// TIA Portal V18 export
DATA_BLOCK "HVAC_Vars"   // DB99
{ S7_Optimized_Access := 'FALSE' }
VERSION : 0.1
// stored: AutoNumber false, DBAccessibleFromOPCUA true, IsOnlyStoredInLoadMemory false, IsWriteProtectedInAS false
   VAR
      Season { S7_SetPoint := 'True'} : "UDT_Store_Season";
      SetPoints { S7_SetPoint := 'True'} : "UDT_Store_Setpoints";
      OpModes { S7_SetPoint := 'True'} : "UDT_Store_OpMode";
      WeekScheduler { S7_SetPoint := 'True'} : "UDT_Store_Scheduler";
      RoomTempSetPointforHMI { S7_SetPoint := 'True'} : Real := 35.0;
      Holidays { S7_SetPoint := 'True'} : Array[1..4] of Date;
      xIsHoliday : Bool := FALSE;
      cDayType : Byte := 16#01;   // 0-WD,1-Mon,2-Cуб,3-Нед,4-Свят
      CurrentDate : Date := D#2026-04-20;
      CurrentTOD : Time_Of_Day := TOD#22:03:20.160;
      iRetVal : Int := 1;
   END_VAR
BEGIN
   Season.cSeasonModeSelection := 16#00;
   Season.cActual := 16#00;   // 0 = Summer 1 = Winter 2 = Midseason, 3=Auro
   Season.cTarget := 16#00;
   Season.cReserve := 16#00;
   Season.rOATtoWinter := 10.0;
   Season.rOATtoSummer := 12.0;
   SetPoints.Room.Actual.rRATHeating := 5.0;
   SetPoints.Room.Actual.rRATCooling := 35.0;
   SetPoints.Room.Actual.rIAQ := 0.0;
   SetPoints.Room.Actual.rBuildingdP := 0.0;
   SetPoints.Room.Comfort.rRATHeating := 18.0;
   SetPoints.Room.Comfort.rRATCooling := 22.0;
   SetPoints.Room.Comfort.rIAQ := 600.0;
   SetPoints.Room.Comfort.rBuildingdP := 5.0;
   SetPoints.Room.PreComfort.rRATHeating := 16.0;
   SetPoints.Room.PreComfort.rRATCooling := 25.0;
   SetPoints.Room.PreComfort.rIAQ := 800.0;
   SetPoints.Room.PreComfort.rBuildingdP := 2.0;
   SetPoints.Room.Econom.rRATHeating := 15.0;
   SetPoints.Room.Econom.rRATCooling := 30.0;
   SetPoints.Room.Econom.rIAQ := 0.0;
   SetPoints.Room.Econom.rBuildingdP := 0.0;
   SetPoints.Room.Protection.rRATHeating := 5.0;
   SetPoints.Room.Protection.rRATCooling := 35.0;
   SetPoints.Room.Protection.rIAQ := 0.0;
   SetPoints.Room.Protection.rBuildingdP := 0.0;
   OpModes.cPreviousOne := 16#00;
   OpModes.cActual := 16#00;
   OpModes.cTarget := 16#00;
   OpModes.cPreselectedOpMode := 16#00;
   WeekScheduler.cOpModeNowByScheduler := 16#02;   // 0 - Prot/ 1-Eco/ 2-PreComf/ 3- Comf/ 4 - Auto
   WeekScheduler.Monday.Comfort.Start := TOD#06:00:00;
   WeekScheduler.Monday.Comfort.Stop := TOD#21:00:00;
   WeekScheduler.Monday.PreComfort.Start := TOD#04:00:00;
   WeekScheduler.Monday.PreComfort.Stop := TOD#23:59:59;
   WeekScheduler.WorkingDays.Comfort.Start := TOD#06:00:00;
   WeekScheduler.WorkingDays.Comfort.Stop := TOD#21:00:00;
   WeekScheduler.WorkingDays.PreComfort.Start := TOD#00:00:00;
   WeekScheduler.WorkingDays.PreComfort.Stop := TOD#23:59:59;
   WeekScheduler.Saturday.Comfort.Start := TOD#06:00:00;
   WeekScheduler.Saturday.Comfort.Stop := TOD#21:00:00;
   WeekScheduler.Saturday.PreComfort.Start := TOD#00:00:00;
   WeekScheduler.Saturday.PreComfort.Stop := TOD#22:00:00;
   WeekScheduler.Sunday.Comfort.Start := TOD#06:00:00;
   WeekScheduler.Sunday.Comfort.Stop := TOD#18:00:00;
   WeekScheduler.Sunday.PreComfort.Start := TOD#05:30:00;
   WeekScheduler.Sunday.PreComfort.Stop := TOD#22:00:00;
   WeekScheduler.Holiday.Comfort.Start := TOD#00:00:00;
   WeekScheduler.Holiday.Comfort.Stop := TOD#00:00:00;
   WeekScheduler.Holiday.PreComfort.Start := TOD#00:00:00;
   WeekScheduler.Holiday.PreComfort.Stop := TOD#00:00:00;
   Holidays[1] := D#2026-01-01;
   Holidays[2] := D#2026-04-12;
   Holidays[3] := D#2027-01-01;
END_DATA_BLOCK
